Fanuc KAREL source: ko00053.KL

-- PROVISIONAL review KL for V770-1; original PC SHA256 7a4b8724e816fff5bcaeb0cc76fe4d95ef619df1495a365c7783b58786677f65
-- Incomplete behavior may be omitted. Consult companion uncertainty JSON. Do not deploy.
PROGRAM KO00053
%NOLOCKGROUP
BEGIN
  -- UNRESOLVED_PC offsets 5-12; opcodes 9D,23
  -- UNRESOLVED_PC offsets 17-69; opcodes 27,27,49,7E,AD,27,49,7E,AD,22,31,7E,4A
  -- UNRESOLVED_PC offsets 74-78; opcodes 7F
END KO00053
